Universal Robots PolyScope program: zigzag_run.urp

Program zigzag_run (installation=default directory=/programs/usbdisk createdIn=5.12.4.1101661 lastSavedIn=5.12.4.1101661)
Robot Program (runOnlyOnce=true)
  Script file /programs/usbdisk/zigzag.script
    | def draw_svg():
    |   draw_z = 0.074940
    |   # home
    |   movel(p[0.598550, -0.129200, 0.105150, 2.249000, -2.194000, 0.000000], a=0.8, v=0.25, r=0.0)
    |   # stroke 0 (form id 0): polyline
    |   movel(p[0.756748, -0.269703, 0.118080, 2.230000, -2.212000, 0.000000], a=0.8, v=0.25, r=0.0)
    |   movep(p[0.756748, -0.269703, draw_z, 2.230000, -2.212000, 0.000000], a=0.5, v=0.02, r=0.015000)
    |   movep(p[0.452671, -0.274649, draw_z, 2.230000, -2.212000, 0.000000], a=0.5, v=0.02, r=0.015000)
    |   movep(p[0.451972, 0.030303, draw_z, 2.230000, -2.212000, 0.000000], a=0.5, v=0.02, r=0.015000)
    |   movep(p[0.756049, 0.035249, draw_z, 2.230000, -2.212000, 0.000000], a=0.5, v=0.02, r=0.000000)
    |   movel(p[0.756049, 0.035249, 0.118080, 2.230000, -2.212000, 0.000000], a=0.8, v=0.25, r=0.0)
    |   # park
    |   movel(p[0.598550, -0.129200, 0.105150, 2.249000, -2.194000, 0.000000], a=0.8, v=0.25, r=0.0)
    | end
    | draw_svg()
